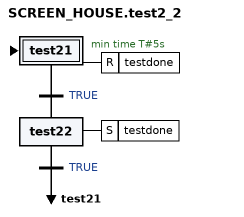
[picture p72: SCREEN_HOUSE.test2_2 (SFC)]
INITIAL_STEP test21: (* min time T#5s *)
	testdone(R);
END_STEP
TRANSITION FROM test21 TO test22 := TRUE;
END_TRANSITION
STEP test22:
	testdone(S);
END_STEP
TRANSITION FROM test22 TO test21 := TRUE;
END_TRANSITION
END_ACTION

(* POU INLET_EQ_PUMP_Prototype, SFC *)
PROGRAM INLET_EQ_PUMP_Prototype
VAR
	EQFloatSensorLO: BOOL;
	EQFLoatSensorOP: BOOL;
	EQFloatSensorHi: BOOL;
	Start_Pump_Done: BOOL;
	StreamLineOverFLow: BOOL;
	SBRFloatSensor: BOOL;
	Act_Stop_Pump_done: BOOL;
	Stop_Pump_done: BOOL;
	EQFLoatSensorDry: BOOL;
	CriticalAlarm_FloatSensorHi : BOOL;
	CriticalAlarm_FloatSensorDRY : BOOL;
	Warning_FloatSensorDry : BOOL;
	Duty_RemoteMode: BOOL;
	Timer1: TON;
	TimerQ: BOOL;
	Duty_Overload: BOOL;
	Duty_Incomplete: BOOL;
	Duty_StartStatus: BOOL;
	Done_StartPumpStandby: BOOL;
	Done_StartStandby: BOOL;
	Done_Start: BOOL;
	Done_Stop: BOOL;
	Done_Timer: BOOL;

	Duty_CommandStart : BOOL;
	Standby_CommandStart: BOOL;
	Standby_RemoteMode: BOOL;
	Standby_Overload: BOOL;
	Standby_Incomplete: BOOL;
	Standby_StartStatus: BOOL;
	Warning_StandbyFailed: BOOL;
	CriticalAlarm_DutyStandbyFailedToStart: BOOL;
	Warning_DutyFailed: BOOL;
	Timer2: TON;
	Done_Timer2: BOOL;
	Timer3: TON;
	Done_Timer3: BOOL;
	Timer4: TON;
	Done_Timer4: BOOL;
	CriticalAlarm_StandbyCannotStop : BOOL;
	CriticalAlarm_DutyCannotStop : BOOL;
	Reset: BOOL;
END_VAR
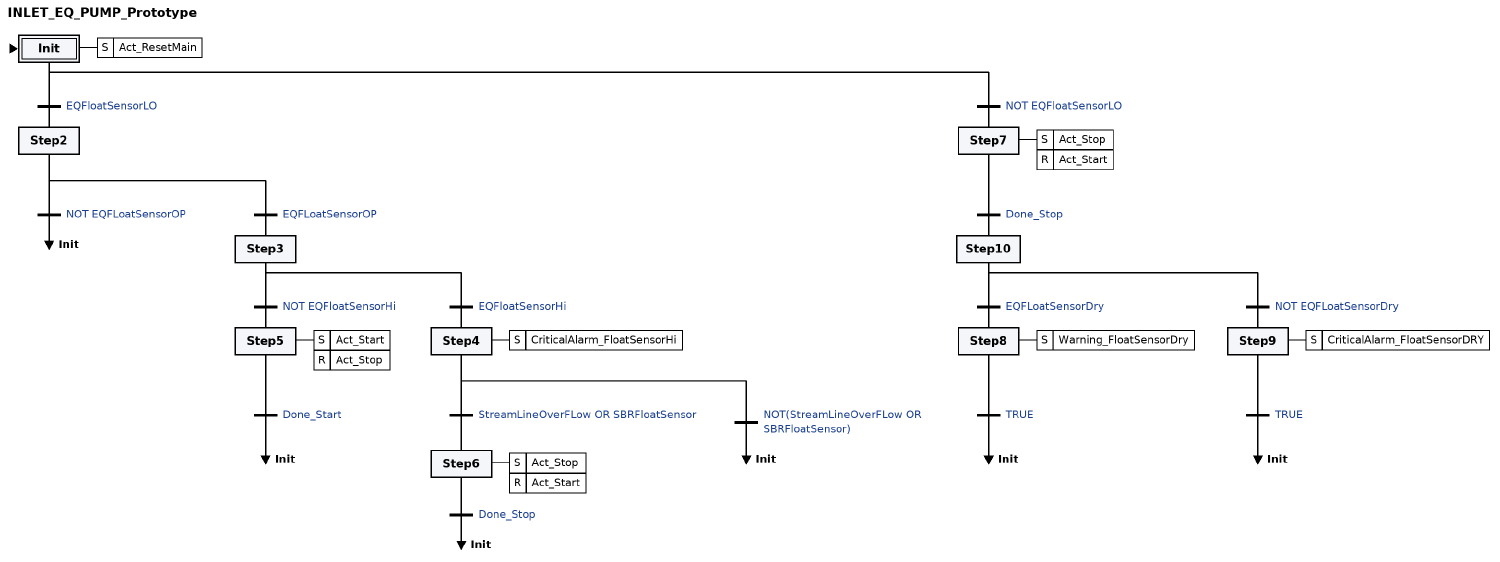
INITIAL_STEP Init:
	Act_ResetMain(S);
END_STEP
TRANSITION FROM Init TO Step2 := EQFloatSensorLO;
END_TRANSITION
TRANSITION FROM Init TO Step7 := NOT EQFloatSensorLO;
END_TRANSITION
STEP Step2:
END_STEP
TRANSITION FROM Step2 TO Init := NOT EQFLoatSensorOP;
END_TRANSITION
TRANSITION FROM Step2 TO Step3 := EQFLoatSensorOP;
END_TRANSITION
STEP Step3:
END_STEP
TRANSITION FROM Step3 TO Step5 := NOT EQFloatSensorHi;
END_TRANSITION
TRANSITION FROM Step3 TO Step4 := EQFloatSensorHi;
END_TRANSITION
STEP Step5:
	Act_Start(S);
	Act_Stop(R);
END_STEP
TRANSITION FROM Step5 TO Init := Done_Start;
END_TRANSITION
STEP Step4:
	CriticalAlarm_FloatSensorHi(S);
END_STEP
TRANSITION FROM Step4 TO Step6 := StreamLineOverFLow OR SBRFloatSensor;
END_TRANSITION
TRANSITION FROM Step4 TO Init := NOT(StreamLineOverFLow OR SBRFloatSensor);
END_TRANSITION
STEP Step6:
	Act_Stop(S);
	Act_Start(R);
END_STEP
TRANSITION FROM Step6 TO Init := Done_Stop;
END_TRANSITION
STEP Step7:
	Act_Stop(S);
	Act_Start(R);
END_STEP
TRANSITION FROM Step7 TO Step10 := Done_Stop;
END_TRANSITION
STEP Step10:
END_STEP
TRANSITION FROM Step10 TO Step8 := EQFLoatSensorDry;
END_TRANSITION
TRANSITION FROM Step10 TO Step9 := NOT EQFLoatSensorDry;
END_TRANSITION
STEP Step8:
	Warning_FloatSensorDry(S);
END_STEP
TRANSITION FROM Step8 TO Init := TRUE;
END_TRANSITION
STEP Step9:
	CriticalAlarm_FloatSensorDRY(S);
END_STEP
TRANSITION FROM Step9 TO Init := TRUE;
END_TRANSITION
END_PROGRAM
ACTION Act_Reset:
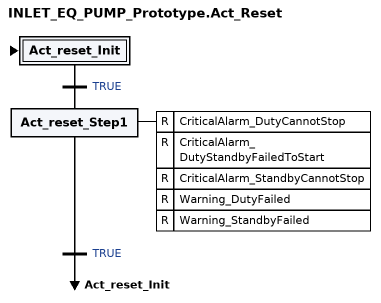
INITIAL_STEP Act_reset_Init:
END_STEP
TRANSITION FROM Act_reset_Init TO Act_reset_Step1 := TRUE;
END_TRANSITION
STEP Act_reset_Step1:
	CriticalAlarm_DutyCannotStop(R);
	CriticalAlarm_DutyStandbyFailedToStart(R);
	CriticalAlarm_StandbyCannotStop(R);
	Warning_DutyFailed(R);
	Warning_StandbyFailed(R);
END_STEP
TRANSITION FROM Act_reset_Step1 TO Act_reset_Init := TRUE;
END_TRANSITION
END_ACTION
ACTION Act_ResetMain:
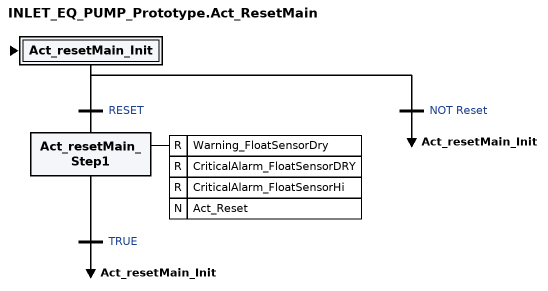
INITIAL_STEP Act_resetMain_Init:
END_STEP
TRANSITION FROM Act_resetMain_Init TO Act_resetMain_Step1 := RESET;
END_TRANSITION
TRANSITION FROM Act_resetMain_Init TO Act_resetMain_Init := NOT Reset;
END_TRANSITION
STEP Act_resetMain_Step1:
	Warning_FloatSensorDry(R);
	CriticalAlarm_FloatSensorDRY(R);
	CriticalAlarm_FloatSensorHi(R);
	Act_Reset(N);
END_STEP
TRANSITION FROM Act_resetMain_Step1 TO Act_resetMain_Init := TRUE;
END_TRANSITION
END_ACTION
ACTION Act_Start:
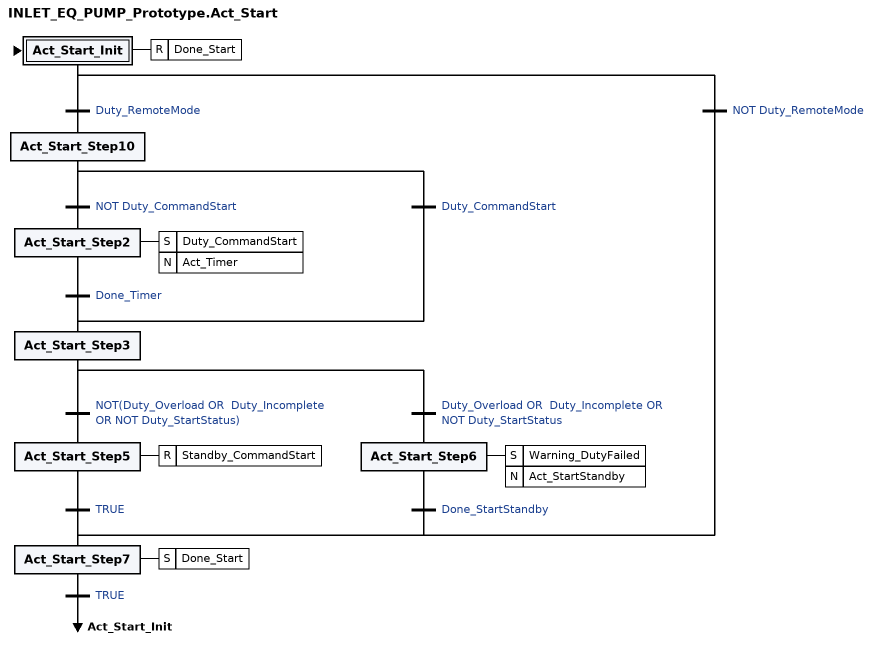
INITIAL_STEP Act_Start_Init:
	Done_Start(R);
END_STEP
TRANSITION FROM Act_Start_Init TO Act_Start_Step10 := Duty_RemoteMode;
END_TRANSITION
TRANSITION FROM Act_Start_Init TO Act_Start_Step7 := NOT Duty_RemoteMode;
END_TRANSITION
STEP Act_Start_Step10:
END_STEP
TRANSITION FROM Act_Start_Step10 TO Act_Start_Step2 := NOT Duty_CommandStart;
END_TRANSITION
TRANSITION FROM Act_Start_Step10 TO Act_Start_Step3 := Duty_CommandStart;
END_TRANSITION
STEP Act_Start_Step2:
	Duty_CommandStart(S);
	Act_Timer(N);
END_STEP
TRANSITION FROM Act_Start_Step2 TO Act_Start_Step3 := Done_Timer;
END_TRANSITION
STEP Act_Start_Step3:
END_STEP
TRANSITION FROM Act_Start_Step3 TO Act_Start_Step5 := NOT(Duty_Overload OR  Duty_Incomplete OR NOT Duty_StartStatus);
END_TRANSITION
TRANSITION FROM Act_Start_Step3 TO Act_Start_Step6 := Duty_Overload OR  Duty_Incomplete OR NOT Duty_StartStatus;
END_TRANSITION
STEP Act_Start_Step5:
	Standby_CommandStart(R);
END_STEP
TRANSITION FROM Act_Start_Step5 TO Act_Start_Step7 := TRUE;
END_TRANSITION
STEP Act_Start_Step6:
	Warning_DutyFailed(S);
	Act_StartStandby(N);
END_STEP
TRANSITION FROM Act_Start_Step6 TO Act_Start_Step7 := Done_StartStandby;
END_TRANSITION
STEP Act_Start_Step7:
	Done_Start(S);
END_STEP
TRANSITION FROM Act_Start_Step7 TO Act_Start_Init := TRUE;
END_TRANSITION
END_ACTION
ACTION Act_StartStandby:
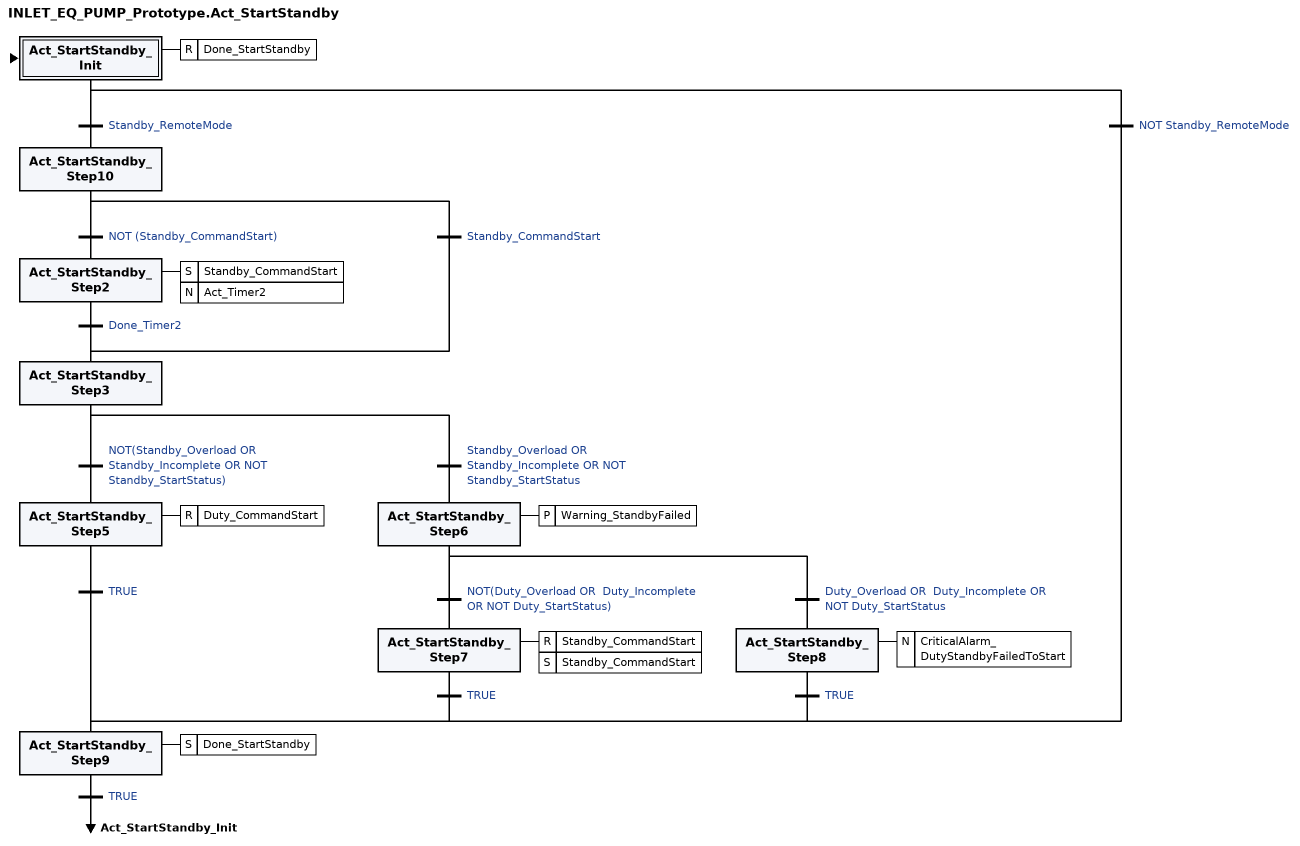
INITIAL_STEP Act_StartStandby_Init:
	Done_StartStandby(R);
END_STEP
TRANSITION FROM Act_StartStandby_Init TO Act_StartStandby_Step10 := Standby_RemoteMode;
END_TRANSITION
TRANSITION FROM Act_StartStandby_Init TO Act_StartStandby_Step9 := NOT Standby_RemoteMode;
END_TRANSITION
STEP Act_StartStandby_Step10:
END_STEP
TRANSITION FROM Act_StartStandby_Step10 TO Act_StartStandby_Step2 := NOT (Standby_CommandStart);
END_TRANSITION
TRANSITION FROM Act_StartStandby_Step10 TO Act_StartStandby_Step3 := Standby_CommandStart;
END_TRANSITION
STEP Act_StartStandby_Step2:
	Standby_CommandStart(S);
	Act_Timer2(N);
END_STEP
TRANSITION FROM Act_StartStandby_Step2 TO Act_StartStandby_Step3 := Done_Timer2;
END_TRANSITION
STEP Act_StartStandby_Step3:
END_STEP
TRANSITION FROM Act_StartStandby_Step3 TO Act_StartStandby_Step5 := NOT(Standby_Overload OR  Standby_Incomplete OR NOT Standby_StartStatus);
END_TRANSITION
TRANSITION FROM Act_StartStandby_Step3 TO Act_StartStandby_Step6 := Standby_Overload OR  Standby_Incomplete OR NOT Standby_StartStatus;
END_TRANSITION
STEP Act_StartStandby_Step5:
	Duty_CommandStart(R);
END_STEP
TRANSITION FROM Act_StartStandby_Step5 TO Act_StartStandby_Step9 := TRUE;
END_TRANSITION
STEP Act_StartStandby_Step6:
	Warning_StandbyFailed(P);
END_STEP
TRANSITION FROM Act_StartStandby_Step6 TO Act_StartStandby_Step7 := NOT(Duty_Overload OR  Duty_Incomplete OR NOT Duty_StartStatus);
END_TRANSITION
TRANSITION FROM Act_StartStandby_Step6 TO Act_StartStandby_Step8 := Duty_Overload OR  Duty_Incomplete OR NOT Duty_StartStatus;
END_TRANSITION
STEP Act_StartStandby_Step7:
	Standby_CommandStart(R);
	Standby_CommandStart(S);
END_STEP
TRANSITION FROM Act_StartStandby_Step7 TO Act_StartStandby_Step9 := TRUE;
END_TRANSITION
STEP Act_StartStandby_Step8:
	CriticalAlarm_DutyStandbyFailedToStart (N);
END_STEP
TRANSITION FROM Act_StartStandby_Step8 TO Act_StartStandby_Step9 := TRUE;
END_TRANSITION
STEP Act_StartStandby_Step9:
	Done_StartStandby(S);
END_STEP
TRANSITION FROM Act_StartStandby_Step9 TO Act_StartStandby_Init := TRUE;
END_TRANSITION
END_ACTION
ACTION Act_Stop:
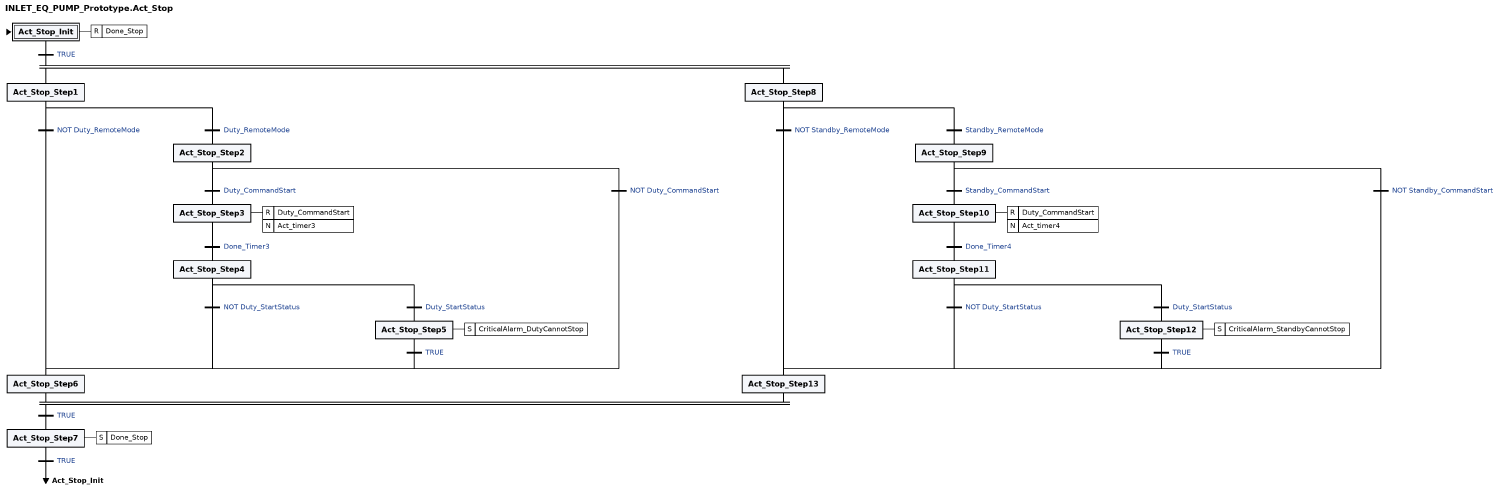
INITIAL_STEP Act_Stop_Init:
	Done_Stop(R);
END_STEP
TRANSITION FROM Act_Stop_Init TO (Act_Stop_Step1, Act_Stop_Step8) := TRUE;
END_TRANSITION
STEP Act_Stop_Step1:
END_STEP
TRANSITION FROM Act_Stop_Step1 TO Act_Stop_Step6 := NOT Duty_RemoteMode;
END_TRANSITION
TRANSITION FROM Act_Stop_Step1 TO Act_Stop_Step2 := Duty_RemoteMode;
END_TRANSITION
STEP Act_Stop_Step2:
END_STEP
TRANSITION FROM Act_Stop_Step2 TO Act_Stop_Step3 := Duty_CommandStart;
END_TRANSITION
TRANSITION FROM Act_Stop_Step2 TO Act_Stop_Step6 := NOT Duty_CommandStart;
END_TRANSITION
STEP Act_Stop_Step3:
	Duty_CommandStart(R);
	Act_timer3(N);
END_STEP
TRANSITION FROM Act_Stop_Step3 TO Act_Stop_Step4 := Done_Timer3;
END_TRANSITION
STEP Act_Stop_Step4:
END_STEP
TRANSITION FROM Act_Stop_Step4 TO Act_Stop_Step6 := NOT Duty_StartStatus;
END_TRANSITION
TRANSITION FROM Act_Stop_Step4 TO Act_Stop_Step5 := Duty_StartStatus;
END_TRANSITION
STEP Act_Stop_Step5:
	CriticalAlarm_DutyCannotStop(S);
END_STEP
TRANSITION FROM Act_Stop_Step5 TO Act_Stop_Step6 := TRUE;
END_TRANSITION
STEP Act_Stop_Step6:
END_STEP
STEP Act_Stop_Step8:
END_STEP
TRANSITION FROM Act_Stop_Step8 TO Act_Stop_Step13 := NOT Standby_RemoteMode;
END_TRANSITION
TRANSITION FROM Act_Stop_Step8 TO Act_Stop_Step9 := Standby_RemoteMode;
END_TRANSITION
STEP Act_Stop_Step9:
END_STEP
TRANSITION FROM Act_Stop_Step9 TO Act_Stop_Step10 := Standby_CommandStart;
END_TRANSITION
TRANSITION FROM Act_Stop_Step9 TO Act_Stop_Step13 := NOT Standby_CommandStart;
END_TRANSITION
STEP Act_Stop_Step10:
	Duty_CommandStart(R);
	Act_timer4(N);
END_STEP
TRANSITION FROM Act_Stop_Step10 TO Act_Stop_Step11 := Done_Timer4;
END_TRANSITION
STEP Act_Stop_Step11:
END_STEP
TRANSITION FROM Act_Stop_Step11 TO Act_Stop_Step13 := NOT Duty_StartStatus;
END_TRANSITION
TRANSITION FROM Act_Stop_Step11 TO Act_Stop_Step12 := Duty_StartStatus;
END_TRANSITION
STEP Act_Stop_Step12:
	CriticalAlarm_StandbyCannotStop(S);
END_STEP
TRANSITION FROM Act_Stop_Step12 TO Act_Stop_Step13 := TRUE;
END_TRANSITION
STEP Act_Stop_Step13:
END_STEP
TRANSITION FROM (Act_Stop_Step6, Act_Stop_Step13) TO Act_Stop_Step7 := TRUE;
END_TRANSITION
STEP Act_Stop_Step7:
	Done_Stop(S);
END_STEP
TRANSITION FROM Act_Stop_Step7 TO Act_Stop_Init := TRUE;
END_TRANSITION
END_ACTION
ACTION Act_Timer:
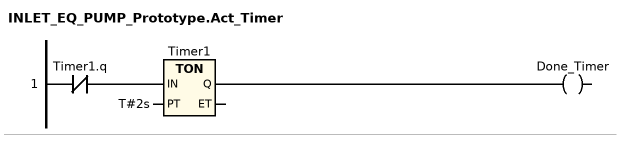
_LD_ (* Ladder Diagram *)
NETWORK 1
	[/Timer1.q] - Timer1:TON(IN: *, PT: T#2s) --- (Done_Timer)
_END_LD_
(* the same logic as Structured Text *)
(* Network 1 *)
Timer1(IN := NOT Timer1.q, PT := T#2s);
Done_Timer := Timer1.Q;
END_ACTION
ACTION Act_Timer2:
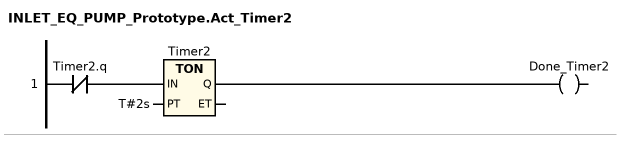
_LD_ (* Ladder Diagram *)
NETWORK 1
	[/Timer2.q] - Timer2:TON(IN: *, PT: T#2s) --- (Done_Timer2)
_END_LD_
(* the same logic as Structured Text *)
(* Network 1 *)
Timer2(IN := NOT Timer2.q, PT := T#2s);
Done_Timer2 := Timer2.Q;
END_ACTION
ACTION Act_Timer3:
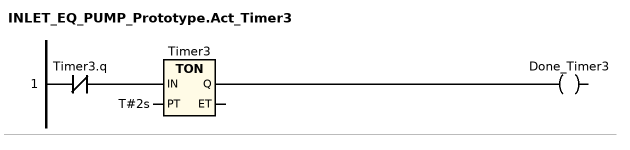
_LD_ (* Ladder Diagram *)
NETWORK 1
	[/Timer3.q] - Timer3:TON(IN: *, PT: T#2s) --- (Done_Timer3)
_END_LD_
(* the same logic as Structured Text *)
(* Network 1 *)
Timer3(IN := NOT Timer3.q, PT := T#2s);
Done_Timer3 := Timer3.Q;
END_ACTION
ACTION Act_Timer4:
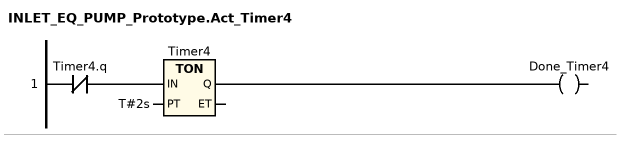
_LD_ (* Ladder Diagram *)
NETWORK 1
	[/Timer4.q] - Timer4:TON(IN: *, PT: T#2s) --- (Done_Timer4)
_END_LD_
(* the same logic as Structured Text *)
(* Network 1 *)
Timer4(IN := NOT Timer4.q, PT := T#2s);
Done_Timer4 := Timer4.Q;
END_ACTION
